FUNCTION_BLOCK FB_Calculate IMPLEMENTS I_Calculate
VAR
	{attribute  'hide'}
	lResult : LREAL := 0;
END_VAR


METHOD Clear : I_Calculate
MEMSET(destAddr:= ADR(lResult),fillByte :=0, n:=SIZEOF(lResult));
Clear := THIS^;
END_METHOD


METHOD DecreaseBy : I_Calculate
VAR_INPUT
	lDecreaseBy : REAL;
END_VAR
lResult := lResult - lDecreaseBy;
DecreaseBy := THIS^;
END_METHOD


METHOD DivideBy : I_Calculate
VAR_INPUT
	lDivideBy : REAL;
END_VAR
IF lDivideBy = 0 THEN
	lResult := 0;
ELSE	
	lResult := lResult / lDivideBy;
END_IF

DivideBy := THIS^;
END_METHOD


METHOD GetResult : LREAL
GetResult := lResult;
END_METHOD

METHOD IncreaseBy : I_Calculate
VAR_INPUT
	lIncreaseBy : REAL;
END_VAR
lResult := lResult + lIncreaseBy;
IncreaseBy := THIS^;
END_METHOD


METHOD MultiplyBy : I_Calculate
VAR_INPUT
	lMultiplyBy : REAL;
END_VAR
lResult := lResult * lMultiplyBy;
MultiplyBy := THIS^;
END_METHOD

METHOD SetNumber : I_Calculate
VAR_INPUT
	lNumber : LREAL;
END_VAR
lResult := lNumber;
SetNumber := THIS^;
END_METHOD

END_FUNCTION_BLOCK

(* stored: Version 1.1.0.1, ProductVersion 3.1.4024.12
   POU FB_Calculate: Id {fd0f0c21-0296-466b-abff-e0b229984285}, SpecialFunc None
   Method Clear: Id {33b45ed3-12a4-4213-8e47-d19c93bca373}
   Method DecreaseBy: Id {6b72b71c-27c8-4bf6-a884-8f4d65f2ba98}
   Method DivideBy: Id {4f10380e-fa29-4ad3-86e5-a4e15fbb69ff}
   Method GetResult: Id {ed0383b5-a43c-41e3-8070-9451dbf58f49}
   Method IncreaseBy: Id {7e263cec-5197-47d7-a28d-e3fc97c94677}
   Method MultiplyBy: Id {0f8b7f56-e647-4043-b82c-156f134385a4}
   Method SetNumber: Id {e56ecddd-c17f-4c0c-b3ed-ea2c5a33467e} *)
